PROGRAM MAIN
VAR
	
    fPotmeter: INT := 0; // Gemeten waarde van potentiometer (0 tot 32767)
    bValue: BYTE; // Geconverteerde waarde (0 tot 15)

END_VAR

bValue := TO_BYTE((fPotmeter * 15) / 32767);

END_PROGRAM

(* stored: Version 1.1.0.1, ProductVersion 3.1.4024.12
   POU MAIN: Id {716b76db-7100-4c9a-91e3-d41f663d3103}, SpecialFunc None *)
